(* CoDeSys 2.3 export: FF_DRE.EXP *)

(* POU Logic/FF edge triggered/FF_DRE, ST *)
FUNCTION_BLOCK FF_DRE
VAR_INPUT
	SET : BOOL;
	D : BOOL;
	CLK : BOOL;
	RST : BOOL;
END_VAR
VAR_OUTPUT
	Q : BOOL;
END_VAR
VAR
	edge : BOOL;
END_VAR


(*
version 1.2	30. oct. 2008
programmer 	hugo
tested by	oscat

D-type flip flop with set, reset and rising clock trigger

*)
IF rst OR set THEN
	Q := NOT rst;
ELSIF clk AND NOT edge THEN
	Q := D;
END_IF;
edge := CLK;

(* revision history
hm	4. aug 2006		rev 1.0
	original version

hm	27. dec 2007	rev 1.1
	changed code for better performance

hm	30. oct. 2008	rev 1.2
	optimized performance
*)
END_FUNCTION_BLOCK
